Fanuc KAREL source: kc00009.KL

-- PROVISIONAL review KL for V770-1; original PC SHA256 648f65c15b797689e9347feaab6038d12027e4a99e6155e23376300c3e97b475
-- Incomplete behavior may be omitted. Consult companion uncertainty JSON. Do not deploy.
PROGRAM KC00009
%NOLOCKGROUP
BEGIN
  -- UNRESOLVED_PC offsets 5-33; opcodes 27,22,1C,22,22,31
  -- UNRESOLVED_PC offsets 38-42; opcodes 7F
END KC00009
